FUNCTION_BLOCK Conveyor EXTENDS BaseComponent
VAR_INPUT
END_VAR
VAR_OUTPUT
END_VAR
VAR
	Motor : Motor;
END_VAR

METHOD METH_ConveyorBackward : BOOL
VAR_INPUT
END_VAR
Motor.ACT_TurnCounterclockwise();
END_METHOD

METHOD METH_ConveyorForward : BOOL
VAR_INPUT
END_VAR
Motor.ACT_TurnClockwise();
END_METHOD

METHOD METH_ConveyorStop : BOOL
VAR_INPUT
END_VAR
Motor.ACT_Stop();
END_METHOD

END_FUNCTION_BLOCK

(* stored: Version 1.1.0.1
   POU Conveyor: Id {ec7bb8df-4121-4927-8bcd-202c4b16387c}, SpecialFunc None
   Method METH_ConveyorBackward: Id {39684807-ecc3-45bb-919f-174939b78c07}
   Method METH_ConveyorForward: Id {cba2b1c1-0e88-4be7-90e1-04ceb0d1198e}
   Method METH_ConveyorStop: Id {4443a639-c5bb-4dff-9f71-d719fc932092} *)
